(* PLC project Generated.project, CODESYS CODESYS V3.5 SP19 Patch 1 *)
(* stored: creationDateTime 2026-09-01T00:57:57.914330, modificationDateTime 2026-09-01T00:57:57.914330 *)

(* ═══════════════════════════════════════════════════════════════ 🚦 ST_CycleDumpAtTremieState — États publics cycle vidage trémie (legacy) ═══════════════════════════════════════════════════════════════ *)
TYPE ST_CycleDumpAtTremieState : STRUCT
  DumpAtTremieArmed : BOOL;  (* TglEnableDumpAtTremie (bit IHM brut) *)
  DumpAtTremieAssistActive : BOOL;  (* Armé ET Mode MAINT_N1/N2 (mode réellement actif) *)
  DumpAtTremieAtTremie : BOOL;  (* M3_AtTremieStable *)
  DumpAtTremieBucketOpenArmed : BOOL;  (* CmdOpen_IHM déclenché par ce mode *)
  DumpAtTremieDescentLocked : BOOL;  (* DescendPermit M1/M2 forcé par ce mode (hors P1/Maintenance) *)
END_STRUCT;
END_TYPE
